INTERFACE I_TestResults

METHOD GetAreTestResultsAvailable : BOOL
END_METHOD

METHOD GetTestSuiteResults : REFERENCE TO ST_TestSuiteResults
END_METHOD

END_INTERFACE

(* stored: Version 1.1.0.1, ProductVersion 3.1.4022.18
   Itf I_TestResults: Id {4b8dc1ed-f636-46c0-8e7c-15c7836626f3}
   Method GetAreTestResultsAvailable: Id {28adb76a-ca7f-4d42-9fad-44627006532d}
   Method GetTestSuiteResults: Id {f78f0f3e-a842-41e1-b891-bfd5e3fc0531} *)
